ABB RobotStudio station: Proiect_Robotica_Drapiciuc_Munteanu.rspag

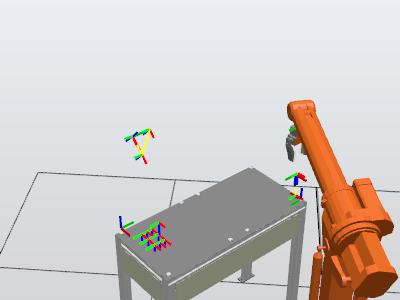
--- station ---
Station Project5 (saved by RobotStudio 22.3.10190.2)
Controller Controller6
  mechanical unit ROB_1: IRB1400_5_144__01, 6 joints, base frame (0, 0, 0) mm
Layout (positions relative to the parent item):
  - IRB1400_5_144__01 [mechanism, from Robots\IRB1400_5_144__01.rslib] at (0, 0, 0) mm; joint values [-1.2898, 0.0063, -0.1877, 0, 1.7586, -0.5043] (rad or m)
  - Gripper_R1400 [smart component, from Components\Gripper_R1400.rslib] at (232.62, -805.83, 1242.2) mm, rotated rx 180 ry -0.01 rz 134.99 deg
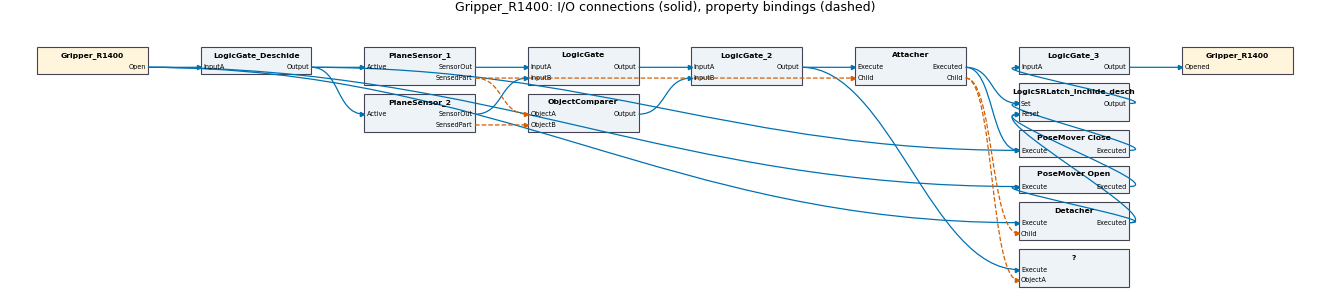
      connections:
        Attacher.Executed -> LogicSRLatch_Inchide_deschide.Set
        Detacher.Executed -> LogicSRLatch_Inchide_deschide.Reset
        Attacher.Executed -> PoseMover Close.Execute
        PoseMover Close.Executed -> LogicSRLatch_Inchide_deschide.Set
        Detacher.Executed -> PoseMover Open.Execute
        PoseMover Open.Executed -> LogicSRLatch_Inchide_deschide.Reset
        LogicGate.Output -> LogicGate_2.InputA
        ObjectComparer.Output -> LogicGate_2.InputB
        LogicGate_2.Output -> ?.Execute
        LogicGate_2.Output -> Attacher.Execute
        PlaneSensor_1.SensorOut -> LogicGate.InputA
        PlaneSensor_2.SensorOut -> LogicGate.InputB
        LogicGate_Deschide.Output -> PlaneSensor_2.Active
        LogicGate_Deschide.Output -> PlaneSensor_1.Active
        LogicGate_Deschide.Output -> PoseMover Close.Execute
        LogicSRLatch_Inchide_deschide.Output -> LogicGate_3.InputA
        LogicGate_3.Output -> Gripper_R1400.Opened
        Gripper_R1400.Open -> LogicGate_Deschide.InputA
        Gripper_R1400.Open -> Detacher.Execute
        Gripper_R1400.Open -> PoseMover Open.Execute
        Attacher.Child => Detacher.Child
        Attacher.Child => ?.ObjectA
        PlaneSensor_1.SensedPart => Attacher.Child
        PlaneSensor_1.SensedPart => ObjectComparer.ObjectA
        PlaneSensor_2.SensedPart => ObjectComparer.ObjectB
    - Attacher [smart component, from Components\Gripper_R1400.rslib]
        properties: Parent=Gripper; Flange=0; Child=(none); Mount=false; Offset=[0 0 0]; Orientation=[0 0 0]
    - Detacher [smart component, from Components\Gripper_R1400.rslib]
        properties: Child=(none); KeepPosition=true
    - LogicGate_Deschide [smart component, from Components\Gripper_R1400.rslib]
        properties: Operator=NOT; Delay=0
    - LogicSRLatch_Inchide_deschide [smart component, from Components\Gripper_R1400.rslib]
    - PoseMover Close [smart component, from Components\Gripper_R1400.rslib]
        properties: Mechanism=Gripper; Pose=3; Duration=0
    - PoseMover Open [smart component, from Components\Gripper_R1400.rslib]
        properties: Mechanism=Gripper; Pose=2; Duration=0
    - ObjectComparer [smart component, from Components\ObjectComparer.rslib]
        properties: ObjectA=(none); ObjectB=(none)
    - LogicGate [smart component, from Components\LogicGate.rslib]
        properties: Operator=AND; Delay=0
    - LogicGate_2 [smart component, from Components\LogicGate.rslib]
        properties: Operator=AND; Delay=0
    - PlaneSensor_1 [smart component, from Components\PlaneSensor.rslib]
        properties: Origin=[-0.015 0.03 0.128]; Axis1=[0 0 0.055]; Axis2=[0.03 0 0]; SensedPart=(none)
      - _sensorPart_ [part], size 30 x 0 x 55 mm
    - PlaneSensor_2 [smart component, from Components\PlaneSensor.rslib]
        properties: Origin=[-0.015 -0.03 0.128]; Axis1=[0 0 0.055]; Axis2=[0.03 0 0]; SensedPart=(none)
      - _sensorPart_ [part], size 30 x 0 x 55 mm
    - Gripper [mechanism, from Components\Gripper_R1400.rslib] at (0, 0.03, 0) mm; joint values [0, 0] (rad or m)
    - LogicGate_3 [smart component, from Components\LogicGate.rslib]
        properties: Operator=NOT; Delay=0
  - Stoc1400 [smart component, from Components\Stoc1400.rslib] at (629.33, -613.77, 0) mm, rotated rx 0 ry 0 rz 135 deg
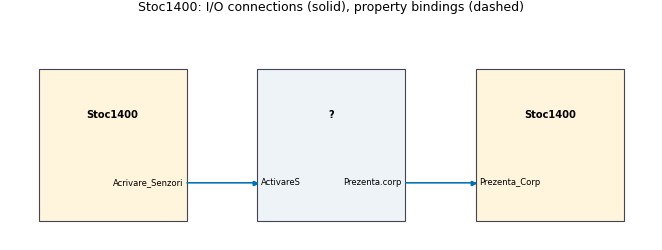
      connections:
        Stoc1400.Acrivare_Senzori -> ?.ActivareS
        Stoc1400.Acrivare_Senzori -> ?.ActivareS
        ?.Prezenta.corp -> Stoc1400.Prezenta_Corp
        ?.Prezenta.corp -> Stoc1400.Prezenta_Corp
    - 679#Body 1 [part, from Components\Stoc1400.rslib]
    - 681#Body 2 [part, from Components\Stoc1400.rslib]
    - 683#Body 3 [part, from Components\Stoc1400.rslib]
    - 685#Body 4 [part, from Components\Stoc1400.rslib]
    - 687#Body 5 [part, from Components\Stoc1400.rslib]
    - 689#Body 6 [part, from Components\Stoc1400.rslib]
    - 691#Body 7 [part, from Components\Stoc1400.rslib]
    - 693#Body 8 [part, from Components\Stoc1400.rslib]
    - 695#Body 9 [part, from Components\Stoc1400.rslib]
    - 697#Body 10 [part, from Components\Stoc1400.rslib]
    - 701#Body 12 [part, from Components\Stoc1400.rslib]
    - 703#Body 13 [part, from Components\Stoc1400.rslib]
    - 705#Body 14 [part, from Components\Stoc1400.rslib]
    - 707#Body 15 [part, from Components\Stoc1400.rslib]
    - 755#Body 39 [part, from Components\Stoc1400.rslib]
    - 757#Body 40 [part, from Components\Stoc1400.rslib]
    - 759#Body 41 [part, from Components\Stoc1400.rslib]
    - 761#Body 42 [part, from Components\Stoc1400.rslib]
    - 785#Body 54 [part, from Components\Stoc1400.rslib]
    - 787#Body 55 [part, from Components\Stoc1400.rslib]
    - 789#Body 56 [part, from Components\Stoc1400.rslib]
    - 791#Body 57 [part, from Components\Stoc1400.rslib]
    - 793#Body 58 [part, from Components\Stoc1400.rslib]
    - Part [part, from Components\Stoc1400.rslib]
    - Part_2 [part, from Components\Stoc1400.rslib]
    - Part_3 [part, from Components\Stoc1400.rslib]
    - Part_4 [part, from Components\Stoc1400.rslib]
  - Positioner_piesa [smart component, from Components\Positioner.rslib]
      properties: Object=(none); Position=[0.410122 -0.8754 0.82]; Orientation=[0 0 -2.35619449019234]; Reference=Global; ReferenceObject=(none)
  - Attacher_piesa [smart component, from Components\Attacher.rslib]
      properties: Parent=Gripper_R1400; Flange=0; Child=(none); Mount=false; Offset=[0 0 0]; Orientation=[0 0 0]
  - Detacher_piesa [smart component, from Components\Detacher.rslib]
      properties: Child=(none); KeepPosition=true
  - Frame_5 [frame]
Attachment: Gripper_R1400 is attached to IRB1400_5_144__01 / Link6
Station signals: DI piesa_A_positioner
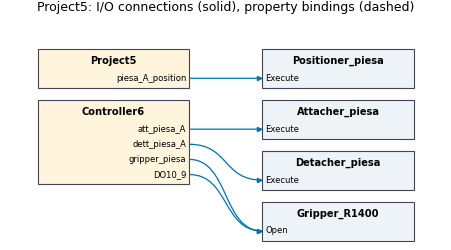
Station logic (signal -> signal, property => property):
  Project5.piesa_A_positioner -> Positioner_piesa.Execute
  Controller6.att_piesa_A -> Attacher_piesa.Execute
  Controller6.dett_piesa_A -> Detacher_piesa.Execute
  Controller6.gripper_piesa -> Gripper_R1400.Open
  Controller6.DO10_9 -> Gripper_R1400.Open
Targets, tools, work objects and paths stored in the station and not in the controller backup, written as RAPID:
! task T_ROB1
MODULE Module1
  CONST robtarget J_M:=[[200,80,0],[0,1,0,0],[-1,-1,0,0],[9E+09,9E+09,9E+09,9E+09,9E+09,9E+09]];
  PROC N()
    MoveL Air,v300,fine,Efector\WObj:=Coords;
    MoveL Jst,v300,fine,Efector\WObj:=Coords;
    MoveL Sst,v300,fine,Efector\WObj:=Coords;
    MoveL Jdr,v300,fine,Efector\WObj:=Coords;
    MoveL Sdr,v300,fine,Efector\WObj:=Coords;
    MoveL Air,v300,fine,Efector\WObj:=Coords;
  ENDPROC
  PROC A()
    MoveL Air,v300,fine,Efector\WObj:=Coords;
    MoveL Jst,v300,fine,Efector\WObj:=Coords;
    MoveL S_M,v300,fine,Efector\WObj:=Coords;
    MoveL Jdr,v300,fine,Efector\WObj:=Coords;
    MoveL JM,v300,fine,Efector\WObj:=Coords;
    MoveL st_M,v300,fine,Efector\WObj:=Coords;
    MoveL dr_M,v300,fine,Efector\WObj:=Coords;
    MoveL Air,v300,fine,Efector\WObj:=Coords;
  ENDPROC
  PROC D()
    MoveL Air,v300,fine,Efector\WObj:=Coords;
    MoveL Sst,v300,fine,Efector\WObj:=Coords;
    MoveL Jst,v300,fine,Efector\WObj:=Coords;
    MoveC dr_M,Sst,v300,fine,Efector\WObj:=Coords;
    MoveL Air,v300,fine,Efector\WObj:=Coords;
  ENDPROC
  PROC Path_10()
    MoveL p30,v300,fine,Efector\WObj:=wobj0;
    MoveL p40,v300,fine,Efector\WObj:=wobj0;
    MoveL p50,v300,fine,Efector\WObj:=wobj0;
  ENDPROC
ENDMODULE


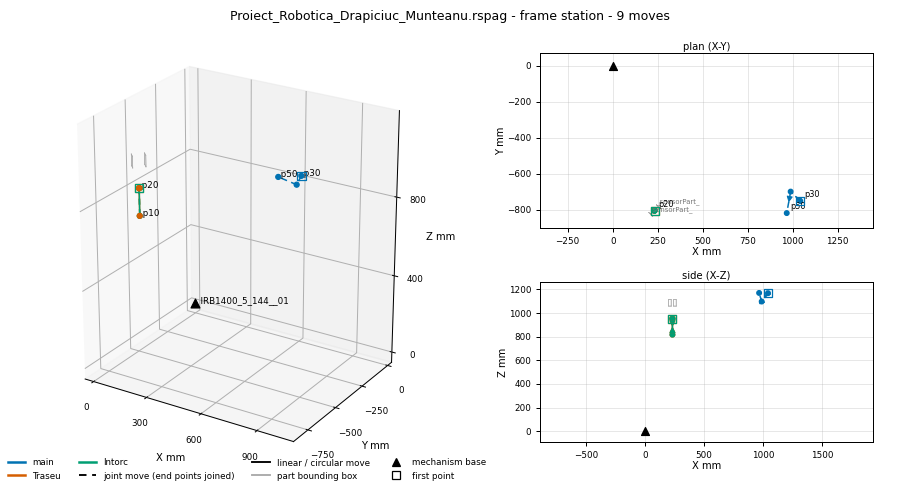
[picture p0: tool path of Proiect_Robotica_Drapiciuc_Munteanu.rspag in frame station, 9 of 29 moves have a stored position in this frame; points joined in program order, loops and branches not executed]
--- Controller Data/Controller6/RAPID/TASK1/PROGMOD/Module1.mod ---
MODULE Module1
    CONST robtarget p20:=[[40.76,9.22,139.9],[5.9E-05,-5E-05,-1,-1.2E-05],[-1,-1,-1,0],[9E+09,9E+09,9E+09,9E+09,9E+09,9E+09]];
    CONST robtarget p10:=[[40.72,9.23,4.9],[8.8E-05,-3.7E-05,-1,-1.7E-05],[-1,-1,-1,0],[9E+09,9E+09,9E+09,9E+09,9E+09,9E+09]];
    CONST robtarget p50:=[[966.601467189,-819.466701626,1170.69],[0.362316816,0.358110668,0.855308085,-0.094505844],[-1,0,0,0],[9E+09,9E+09,9E+09,9E+09,9E+09,9E+09]];
    CONST robtarget p40:=[[988.267446486,-700.10711826,1097.87],[0.362456749,0.358176788,0.855216853,-0.094544323],[-1,-1,0,0],[9E+09,9E+09,9E+09,9E+09,9E+09,9E+09]];
    CONST robtarget p30:=[[1041.979177276,-752.730107301,1168.85],[0.36261717,0.358162943,0.855149453,-0.094591263],[-1,-1,0,0],[9E+09,9E+09,9E+09,9E+09,9E+09,9E+09]];
    CONST robtarget Tag10:=[[945.750262649,-487.904981125,1000.628219509],[-0.000000008,0.382683374,0.923879557,0.000000004],[0,0,-1,0],[9E+09,9E+09,9E+09,9E+09,9E+09,9E+09]];
    CONST robtarget Tag20:=[[478.593921385,-814.862003663,1013.582769169],[0.417934011,0.42537778,0.761953257,-0.252610649],[-1,-1,0,0],[9E+09,9E+09,9E+09,9E+09,9E+09,9E+09]];
    CONST robtarget Tag80:=[[106.668705533,-41.352305249,76.994906394],[0.00536765,-0.431380014,0.902084519,0.011224612],[-1,-1,-1,0],[9E+09,9E+09,9E+09,9E+09,9E+09,9E+09]];
    CONST robtarget Tag40:=[[411.790267154,-880.567704781,822.141824053],[0.026273498,0.3878417,0.921148575,-0.019334491],[-1,0,-1,0],[9E+09,9E+09,9E+09,9E+09,9E+09,9E+09]];
    CONST robtarget Tag802:=[[106.668705533,-41.352305249,76.994906394],[0.00536765,-0.431380014,0.902084519,0.011224612],[-1,-1,-1,0],[9E+09,9E+09,9E+09,9E+09,9E+09,9E+09]];
    CONST robtarget Tag90:=[[26.319905784,177.541247239,82.443122451],[0.00536765,-0.431380014,0.902084519,0.011224612],[-1,-1,-1,0],[9E+09,9E+09,9E+09,9E+09,9E+09,9E+09]];
    CONST robtarget Tag602:=[[26.319905825,179.780635491,-7.529012904],[0.00536765,-0.431380014,0.902084519,0.011224612],[-1,-1,-1,0],[9E+09,9E+09,9E+09,9E+09,9E+09,9E+09]];
    CONST robtarget Tag902:=[[26.319791604,178.356003266,49.708862671],[0.005367642,-0.43138007,0.902084492,0.011224609],[-1,-1,-1,0],[9E+09,9E+09,9E+09,9E+09,9E+09,9E+09]];
    CONST robtarget Tag60:=[[106.668705574,-39.112916997,-12.977228961],[0.00536765,-0.431380014,0.902084519,0.011224612],[-1,-1,-1,0],[9E+09,9E+09,9E+09,9E+09,9E+09,9E+09]];
    PERS tooldata Efector:=[TRUE,[[0,0.033033672,289.3],[1,0,0,0]],[1.5,[0,0,90],[1,0,0,0],0.01,0.01,0.01]];
    PERS wobjdata Wobj2:=[FALSE,TRUE,"",[[460.683469168,-773.537448816,842],[0.66833544,-0.008316079,0.009254535,-0.743755965]],[[0,0,0],[1,0,0,0]]];
    PERS wobjdata Workobject_1:=[FALSE,TRUE,"",[[460.683469168,-773.537448816,842],[0.66833544,-0.008316079,0.009254535,-0.743755965]],[[0,0,0],[1,0,0,0]]];
    PERS wobjdata Workobject_2:=[FALSE,TRUE,"",[[459.619,-1066.317,820],[0.646050022,-0.66007464,-0.253577345,0.287435852]],[[0,0,0],[1,0,0,0]]];
    CONST robtarget Air:=[[200,80,170],[0,1,0,0],[-1,-1,0,0],[9E+09,9E+09,9E+09,9E+09,9E+09,9E+09]];
    CONST robtarget Jst:=[[200,50,0],[0,1,0,0],[-1,-1,0,0],[9E+09,9E+09,9E+09,9E+09,9E+09,9E+09]];
    CONST robtarget Sst:=[[100,50,0],[0,1,0,0],[-1,0,0,0],[9E+09,9E+09,9E+09,9E+09,9E+09,9E+09]];
    CONST robtarget Jdr:=[[200,110,0],[0,1,0,0],[-1,-1,0,0],[9E+09,9E+09,9E+09,9E+09,9E+09,9E+09]];
    CONST robtarget Sdr:=[[100,110,0],[0,1,0,0],[-1,-1,0,0],[9E+09,9E+09,9E+09,9E+09,9E+09,9E+09]];
    PERS wobjdata Coords:=[FALSE,TRUE,"",[[1061.367,-444.064,841.1],[0.382684313,0,0,0.923879168]],[[0,0,0],[1,0,0,0]]];
    CONST robtarget S_M:=[[100,80,0],[0,1,0,0],[-1,-1,0,0],[9E+09,9E+09,9E+09,9E+09,9E+09,9E+09]];
    CONST robtarget JM:=[[150,80,50],[0,1,0,0],[-1,-1,0,0],[9E+09,9E+09,9E+09,9E+09,9E+09,9E+09]];
    CONST robtarget st_M:=[[150,50,0],[0,1,0,0],[-1,-1,0,0],[9E+09,9E+09,9E+09,9E+09,9E+09,9E+09]];
    CONST robtarget dr_M:=[[150,110,0],[0,1,0,0],[-1,-1,0,0],[9E+09,9E+09,9E+09,9E+09,9E+09,9E+09]];
    PERS wobjdata wobj3:=[FALSE,TRUE,"",[[197.283500002,-783.4735,813],[0.923879168,0,0,-0.382684313]],[[0,0,0],[1,0,0,0]]];
    CONST robtarget s_Apuc:=[[335.99892115,850.998768604,120],[0,1,0,0],[-1,-1,-1,0],[9E+09,9E+09,9E+09,9E+09,9E+09,9E+09]];
    CONST robtarget Pix:=[[335.99892115,850.998768604,-20],[0,1,0,0],[-1,-1,-1,0],[9E+09,9E+09,9E+09,9E+09,9E+09,9E+09]];
    PERS wobjdata Tabla:=[FALSE,TRUE,"",[[1039.938744348,-750.731034137,1166.15356987],[0.3616635,-0.330878326,0.16620588,0.855625299]],[[0,0,0],[1,0,0,0]]];
    CONST jointtarget jp1:=[[-100,0,0,0,0,0],[9E9,9E9,9E9,9E9,9E9,9E9]]; !Folosire a tipului de data jointtarget
!***********************************************************
    !
    ! Module:  Module1
    !
    ! Description:
    !   <Insert description here>
    !
    ! Author: Maria-Daniela
    !
    ! Version: 1.0
    !
    !***********************************************************


    !***********************************************************
    !
    ! Procedure main
    !
    !   This is the entry point of your program
    !   Aplicatia are scopul de scriere de catre robot a oricarui sir de caractere formate din literele a,d si n date de la tastatura.
    !***********************************************************
    PROC main()
         MoveAbsJ jp1, v200, z0, tool0\WObj:=wobj0; ! exemplu de folosire a tipului de data jointtarget
         Traseu;
         MoveJ p30,v200,fine,Efector\WObj:=wobj0;
         MoveJ p40,v200,fine,Efector\WObj:=wobj0;
         MoveJ p50,v200,fine,Efector\WObj:=wobj0;
         test2("dan");
         Intorc;
    ENDPROC
    PROC test2(string name)
        var num i:=1;
        WHILE(i<StrLen(name)+1) DO
            IF(StrPart(name,i,1)="d") THEN
                D(i);
                i:=i+1;
            ELSEIF StrPart(name,i,1)="a" THEN
                A(i);
                i:=i+1;
            ELSEIF StrPart(name,i,1)="n" THEN
                N(i);
                i:=i+1;
            ENDIF
        ENDWHILE
    ENDPROC


     PROC N(num i)
        MoveJ RelTool(Air,0,-80*(i-1),0),v200,fine,Efector\WObj:=Tabla;
        MoveJ RelTool(Jst,0,-80*(i-1),0),v200,fine,Efector\WObj:=Tabla;
        MoveJ RelTool(Sst,0,-80*(i-1),0),v200,fine,Efector\WObj:=Tabla;
        MoveJ RelTool(Jdr,0,-80*(i-1),0),v200,fine,Efector\WObj:=Tabla;
        MoveJ RelTool(Sdr,0,-80*(i-1),0),v200,fine,Efector\WObj:=Tabla;
        MoveJ RelTool(Air,0,-80*(i-1),0),v200,fine,Efector\WObj:=Tabla;
    ENDPROC
    PROC A(num i)
        MoveJ RelTool(Air,0,-80*(i-1),0),v200,fine,Efector\WObj:=Tabla;
        MoveJ RelTool(Jst,0,-80*(i-1),0),v200,fine,Efector\WObj:=Tabla;
        MoveJ RelTool(S_M,0,-80*(i-1),0),v200,fine,Efector\WObj:=Tabla;
        MoveJ RelTool(Jdr,0,-80*(i-1),0),v200,fine,Efector\WObj:=Tabla;
        MoveJ RelTool(JM,0,-80*(i-1),0),v200,fine,Efector\WObj:=Tabla;
        MoveJ RelTool(st_M,0,-80*(i-1),0),v200,fine,Efector\WObj:=Tabla;
        MoveJ RelTool(dr_M,0,-80*(i-1),0),v200,fine,Efector\WObj:=Tabla;
        MoveJ RelTool(Air,0,-80*(i-1),0),v200,fine,Efector\WObj:=Tabla;
    ENDPROC
    PROC D(num i)
        MoveJ RelTool(Air,0,-80*(i-1),0),v200,fine,Efector\WObj:=Tabla;
        MoveJ RelTool(Sst,0,-80*(i-1),0),v200,fine,Efector\WObj:=Tabla;
        MoveJ RelTool(Jst,0,-80*(i-1),0),v200,fine,Efector\WObj:=Tabla;
        MoveC RelTool(dr_M,0,-80*(i-1),0),RelTool(Sst,0,-80*(i-1),0),v200,fine,Efector\WObj:=Tabla;
        MoveJ RelTool(Air,0,-80*(i-1),0),v200,fine,Efector\WObj:=Tabla;

    ENDPROC
    PROC Traseu()
        MoveJ p20,v200,fine,Efector\WObj:=wobj3;
        MoveJ p10,v200,fine,Efector\WObj:=wobj3;
        WaitTime 1;
        SetDO DO10_9,0;
        WaitTime 1;
        MoveL p20,v200,fine,Efector\WObj:=wobj3;
    ENDPROC
    PROC Intorc()
        MoveJ p20,v200,fine,Efector\WObj:=wobj3;
        MoveJ p10,v200,fine,Efector\WObj:=wobj3;
        WaitTime 1;
        SetDO DO10_9,1;
        WaitTime 1;
        MoveL p20,v200,fine,Efector\WObj:=wobj3;
    ENDPROC



ENDMODULE

--- Controller Data/Controller6/SYSPAR/EIO.cfg ---
EIO:CFG_1.0:5:60::
#
EIO_BUS:

      -Name "Virtual1"
#
EIO_UNIT_TYPE:

      -Name "Virtual" -VendorName "ABB" -ProductName "Virtual unit"
#
EIO_UNIT:

      -Name "TuIasi" -UnitType "Virtual" -Bus "Virtual1"
#
EIO_SIGNAL:

      -Name "att_piesa_A" -SignalType "DO"

      -Name "dett_piesa_A" -SignalType "DO"

      -Name "gripper_piesa" -SignalType "DO"

      -Name "DO10_9" -SignalType "DO" -Unit "TuIasi" -UnitMap "1" -Access "All"

      -Name "DO11_7" -SignalType "DO" -Unit "TuIasi" -UnitMap "2" -Access "All"

      -Name "DO11_8" -SignalType "DO" -Unit "TuIasi" -UnitMap "3" -Access "All"

      -Name "DO11_9" -SignalType "DO" -Unit "TuIasi" -UnitMap "4" -Access "All"

      -Name "DO12_1" -SignalType "DO" -Unit "TuIasi" -UnitMap "5" -Access "All"

      -Name "DO13_1" -SignalType "DO" -Unit "TuIasi" -UnitMap "7" -Access "All"

      -Name "DI11_9" -SignalType "DI" -Unit "TuIasi" -UnitMap "8" -Access "All"

      -Name "DI13_9" -SignalType "DI" -Unit "TuIasi" -UnitMap "9" -Access "All"

      -Name "AO12_1" -SignalType "AO" -Unit "TuIasi" -UnitMap "16-31"\
      -Access "All"

      -Name "DI12_2" -SignalType "DI" -Unit "TuIasi" -UnitMap "10" -Access "All"

      -Name "DO12_10" -SignalType "DO" -Unit "TuIasi" -UnitMap "11"\
      -Access "All"

      -Name "DI10_1" -SignalType "DI" -Unit "TuIasi" -UnitMap "12" -Access "All"

      -Name "DI10_7" -SignalType "DI" -Unit "TuIasi" -UnitMap "13" -Access "All"

      -Name "DI10_6" -SignalType "DI" -Unit "TuIasi" -UnitMap "14" -Access "All"

      -Name "DI10_5" -SignalType "DI" -Unit "TuIasi" -UnitMap "15" -Access "All"

      -Name "DI10_4" -SignalType "DI" -Unit "TuIasi" -UnitMap "32" -Access "All"

      -Name "DO10_3" -SignalType "DO" -Unit "TuIasi" -UnitMap "33" -Access "All"

      -Name "DO10_4" -SignalType "DO" -Unit "TuIasi" -UnitMap "34" -Access "All"

      -Name "DO10_2" -SignalType "DO" -Unit "TuIasi" -UnitMap "35" -Access "All"

      -Name "DO10_1" -SignalType "DO" -Unit "TuIasi" -UnitMap "36" -Access "All"
#
EIO_ACCESS:

      -Name "All" -Rapid  -LocalManual  -LocalAuto  -RemoteManual  -RemoteAuto
